TYPE ST_Keypad_4x2_Tap :
STRUCT
	Key: ARRAY [0..7] OF ST_DigitalInput;
END_STRUCT
END_TYPE

(* stored: Version 1.1.0.1, ProductVersion 3.1.4024.12
   DUT ST_Keypad_4x2_Tap: Id {060bb48f-f0c1-404a-a1a2-793081abf998} *)
